ADAPTER Adapter_hmi (* Adapter Interface *)
  (* Standard: 61499-1 *)
  (* Version 0.0, 23/09/2021, Pranay Jhunjhunwala, Schneider Electric *)
  PACKAGE Main;
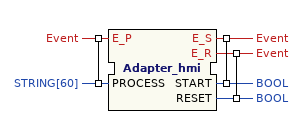
  EVENT_INPUT
    E_P WITH PROCESS; (* Request from Socket *)
  END_EVENT
  EVENT_OUTPUT
    E_S WITH START; (* Confirmation from Plug *)
    E_R WITH RESET; (* Indication from Plug *)
  END_EVENT
  VAR_INPUT
    PROCESS : STRING[60]; (* Request Data from Socket *)
  END_VAR
  VAR_OUTPUT
    START : BOOL; (* Confirmation Data from Plug *)
    RESET : BOOL; (* Indication Data from Plug *)
  END_VAR
  SERVICE SOCKET/PLUG
    SEQUENCE request_confirm
      SOCKET.E_P(PROCESS) -> PLUG.E_P(PROCESS);
      PLUG.E_S(START) -> SOCKET.E_S(START);
    END_SEQUENCE
    SEQUENCE indication_response
      PLUG.E_R(RESET) -> SOCKET.E_R(RESET);
      SOCKET.RSP(RSPD) -> PLUG.RSP(RSPD);
    END_SEQUENCE
  END_SERVICE
END_ADAPTER
